Omron Sysmac Studio project SPA_P8_3 (Sysmac Studio 1.23.0.14, StandardProject)

# Controller new_Controller_0: NX1P2-1040DT1 version 1.18
Axis eje_real, settings changed from default: AxisType=ServoType, UnitsConversion=EnumElement2, UnitsNumerator=8380608, UnitsDenominator=143, MaxVelocity=200, MaxJogVelocity=20, HomingMode=BackupAndPressingTime, StartDirection=NegativeDirection, OriginInputDetectionDirection=NegativeDirection, HomingVelocity=200, HomingApproachVelocity=10, OriginCompensationValue=10, CompensationVelocity=10, ModuloMAXPosition=360, ModuloMINPosition=0, EncoderTypes=Abs
Axis eje_virtual, settings changed from default: AxisNumber=1, UnitsConversion=EnumElement2, UnitsNumerator=8380608, UnitsDenominator=143, MaxVelocity=200, MaxJogVelocity=20
Task PrimaryTask (priority 4, period or condition 2000): Programa0

VAR_GLOBAL CONSTANT
    eje_real : _sAXIS_REF;  (* at MC://_MC_AX[0] *)
END_VAR
VAR_GLOBAL
    PM : BOOL;  (* Pulsador Marcha; at BuiltInIO://cpu/#0/Input_Bit_00 *)
    PP : BOOL;  (* Pulsador Paro; at BuiltInIO://cpu/#0/Input_Bit_01 *)
    PR : BOOL;  (* Pulsador Rearme; at BuiltInIO://cpu/#0/Input_Bit_02 *)
    detector_pieza AT %W0.00 : BOOL;  (* Detector simulado de pieza; published *)
    servo_on AT %W0.01 : BOOL;  (* Interruptor de activación de ejes; published *)
END_VAR
VAR_GLOBAL CONSTANT
    eje_virtual : _sAXIS_REF;  (* at MC://_MC_AX[1] *)
END_VAR
VAR_GLOBAL
    pm_hmi AT %W0.02 : BOOL;  (* Marcha HMI; published *)
    pr_hmi AT %W0.03 : BOOL;  (* Rearme HMI; published *)
    pp_hmi AT %W0.04 : BOOL;  (* Paro HMI; published *)
    pm_var : BOOL;  (* Variable Marcha *)
    pr_var : BOOL;  (* Variable Rearme *)
    pp_var : BOOL;  (* Variable Paro *)
END_VAR
VAR_GLOBAL RETAIN
    piezas_cortadas AT %D0 : INT;  (* Número de piezas cortadas; published *)
END_VAR
VAR_GLOBAL
    detector_negativo : BOOL;  (* Detector de límite negativo; at ECAT://node#2/Digital inputs/NOT *)
    detector_positivo : BOOL;  (* Detector de límite positivo; at ECAT://node#2/Digital inputs/POT *)
    selector_pieza AT %W0.05 : BOOL;  (* ON: 20cm / OFF: 10cm; published *)
END_VAR

PROGRAM Programa0
VAR
    reset_eje_real : MC_Reset;
    power_eje_real : MC_Power;
    home_eje_real : MC_Home;
    etapa_produccion : SINT := 0;  (* Etapa actual grafcet principal *)
    etapa_activar : SINT := 0;  (* Etapa actual grafcet activación *)
    reset_eje_virtual : MC_Reset;
    power_eje_virtual : MC_Power;
    home_eje_virtual : MC_Home;
    inicio_corte : MC_MoveAbsolute;
    grosor_corte : LREAL;  (* Grosor del corte en mm *)
    avance_pieza : MC_MoveRelative;
    retroceso_cinta : MC_MoveZeroPosition;
    corte : MC_MoveRelative;
    MC_inicio_corte : MC_MoveAbsolute;
    MC_corte : MC_MoveRelative;
    cortes_realizados : CTU;
    etapa_paro : SINT;  (* Etapa actual grafcet paro *)
    rearme_cinta : MC_MoveZeroPosition;
    rearme_cortadora : MC_MoveZeroPosition;
    retroceso_cortadora : MC_MoveZeroPosition;
    avance_corte : MC_MoveRelative;
    retroceso_corte : MC_MoveRelative;
    paro_eje_real : MC_Stop;
    paro_eje_virtual : MC_Stop;
    reset_eje_real_paro : MC_Reset;
    reset_eje_virtual_paro : MC_Reset;
    tiempo : BOOL;
    status : _sTimer;
END_VAR
VAR RETAIN
    n_cortes : INT;  (* Número de cortes realizados *)
END_VAR
VAR
    avance_pieza_final : MC_MoveRelative;
    grosor_pieza : LREAL;  (* Grosor de la pieza en mm *)
    grosor_corte_negativo : LREAL;  (* Grosor del corte invertido *)
END_VAR
VAR_EXTERNAL CONSTANT
    eje_real : _sAXIS_REF;
END_VAR
VAR_EXTERNAL
    PM : BOOL;
    servo_on : BOOL;
END_VAR
VAR_EXTERNAL CONSTANT
    eje_virtual : _sAXIS_REF;
END_VAR
VAR_EXTERNAL
    detector_pieza : BOOL;
    PP : BOOL;
    PR : BOOL;
    pm_var : BOOL;
    pm_hmi : BOOL;
    pp_var : BOOL;
    pp_hmi : BOOL;
    pr_var : BOOL;
    pr_hmi : BOOL;
    detector_negativo : BOOL;
    detector_positivo : BOOL;
    selector_pieza : BOOL;
    piezas_cortadas : INT;
END_VAR
VAR
    _p1 : BOOL;
    _e2 : R_TRIG;
    _t3 : BOOL;
END_VAR

(* Section activar: ladder, written here as Structured Text *)

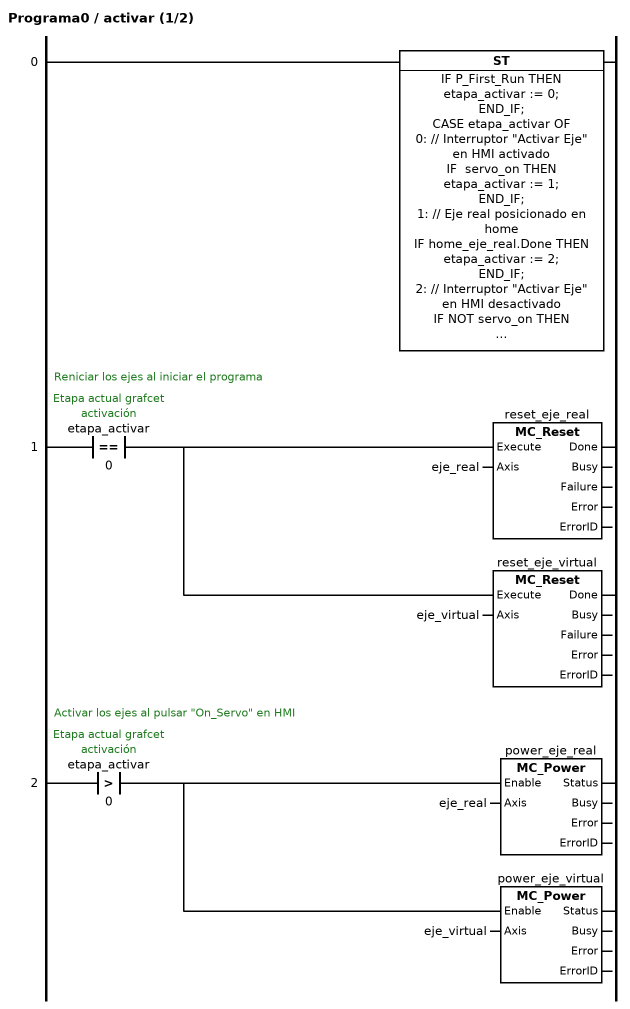
(* Rung 0 *)
IF P_First_Run THEN
	etapa_activar := 0;
END_IF;

CASE etapa_activar OF
	0: // Interruptor "Activar Eje" en HMI activado
		IF  servo_on THEN
			etapa_activar := 1;
		END_IF;
	1: // Eje real posicionado en home
		IF home_eje_real.Done THEN
			etapa_activar := 2;
		END_IF;
	2: // Interruptor "Activar Eje" en HMI desactivado
		IF NOT servo_on THEN
			etapa_activar := 0;
		END_IF;
END_CASE;
(* Rung 1: Reniciar los ejes al iniciar el programa *)
reset_eje_real(Execute := etapa_activar = 0, Axis := eje_real);
reset_eje_virtual(Execute := etapa_activar = 0, Axis := eje_virtual);
(* Rung 2: Activar los ejes al pulsar "On_Servo" en HMI *)
power_eje_real(Enable := etapa_activar > 0, Axis := eje_real);
power_eje_virtual(Enable := etapa_activar > 0, Axis := eje_virtual);

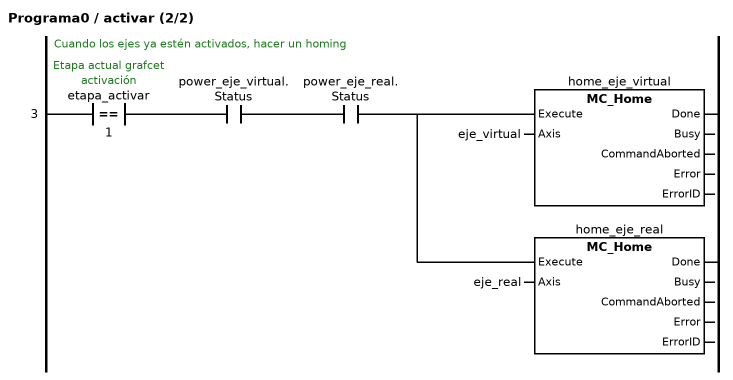
(* Rung 3: Cuando los ejes ya estén activados, hacer un homing *)
_p1 := (etapa_activar = 1) AND power_eje_virtual.Status AND power_eje_real.Status;
home_eje_virtual(Execute := _p1, Axis := eje_virtual);
home_eje_real(Execute := _p1, Axis := eje_real);

(* Section produccion: ladder, written here as Structured Text *)

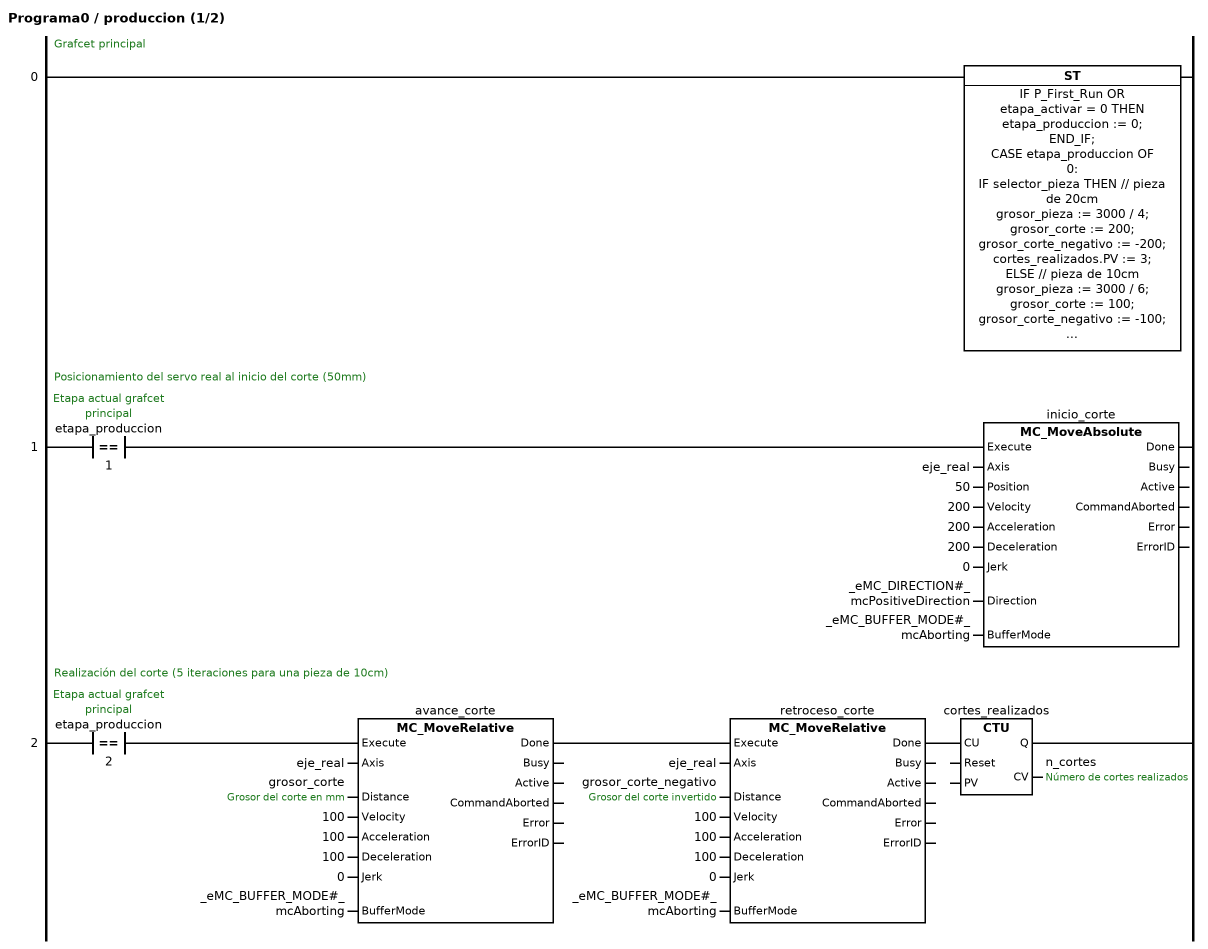
(* Rung 0: Grafcet principal *)
IF P_First_Run OR etapa_activar = 0 THEN
	etapa_produccion := 0;
END_IF;

CASE etapa_produccion OF
    0:
		IF selector_pieza THEN // pieza de 20cm
			grosor_pieza := 3000 / 4;
			grosor_corte := 200;
			grosor_corte_negativo := -200;
			cortes_realizados.PV := 3;
		ELSE // pieza de 10cm
			grosor_pieza := 3000 / 6;
			grosor_corte := 100;
			grosor_corte_negativo := -100;
			cortes_realizados.PV := 5;
		END_IF;
		cortes_realizados.Reset := TRUE;
		// los servos están iniciados y se pulsa marcha
		IF pm_var AND etapa_activar = 2 AND etapa_paro = 0 THEN
			piezas_cortadas := 0;
			cortes_realizados.Reset := FALSE;
			etapa_produccion := 1;
		END_IF;
	1: // el servo real está en posición de inicio de corte (50mm)
		// y se hay pieza en posición de corte
		IF inicio_corte.Done AND detector_pieza THEN
			etapa_produccion := 2;
		END_IF;
	2: // ya se ha realizado el corte de la pieza
		IF retroceso_corte.Done THEN
			piezas_cortadas := piezas_cortadas + 1;
			etapa_produccion := 3;
		END_IF;
	3: // la pieza ya ha avanzado a la posición de corte
		IF cortes_realizados.Q THEN // ya se han realizado todos los cortes
			piezas_cortadas := piezas_cortadas + 1;
			etapa_produccion := 4;
		ELSIF avance_pieza.Done THEN // no se han realizado todos los cortes
			etapa_produccion := 1;
		END_IF;
	4: // la cinta ya ha vuelto al inicio
		IF retroceso_cinta.Done THEN
			etapa_produccion := 0;
		END_IF;
END_CASE;
(* Rung 1: Posicionamiento del servo real al inicio del corte (50mm) *)
inicio_corte(Execute := etapa_produccion = 1, Axis := eje_real, Position := 50, Velocity := 200, Acceleration := 200, Deceleration := 200, Jerk := 0, Direction := _eMC_DIRECTION#_mcPositiveDirection, BufferMode := _eMC_BUFFER_MODE#_mcAborting);
(* Rung 2: Realización del corte (5 iteraciones para una pieza de 10cm) *)
avance_corte(Execute := etapa_produccion = 2, Axis := eje_real, Distance := grosor_corte, Velocity := 100, Acceleration := 100, Deceleration := 100, Jerk := 0, BufferMode := _eMC_BUFFER_MODE#_mcAborting);
retroceso_corte(Execute := avance_corte.Done, Axis := eje_real, Distance := grosor_corte_negativo, Velocity := 100, Acceleration := 100, Deceleration := 100, Jerk := 0, BufferMode := _eMC_BUFFER_MODE#_mcAborting);
_e2(CLK := retroceso_corte.Done);
cortes_realizados(CU := _e2.Q, CV => n_cortes);

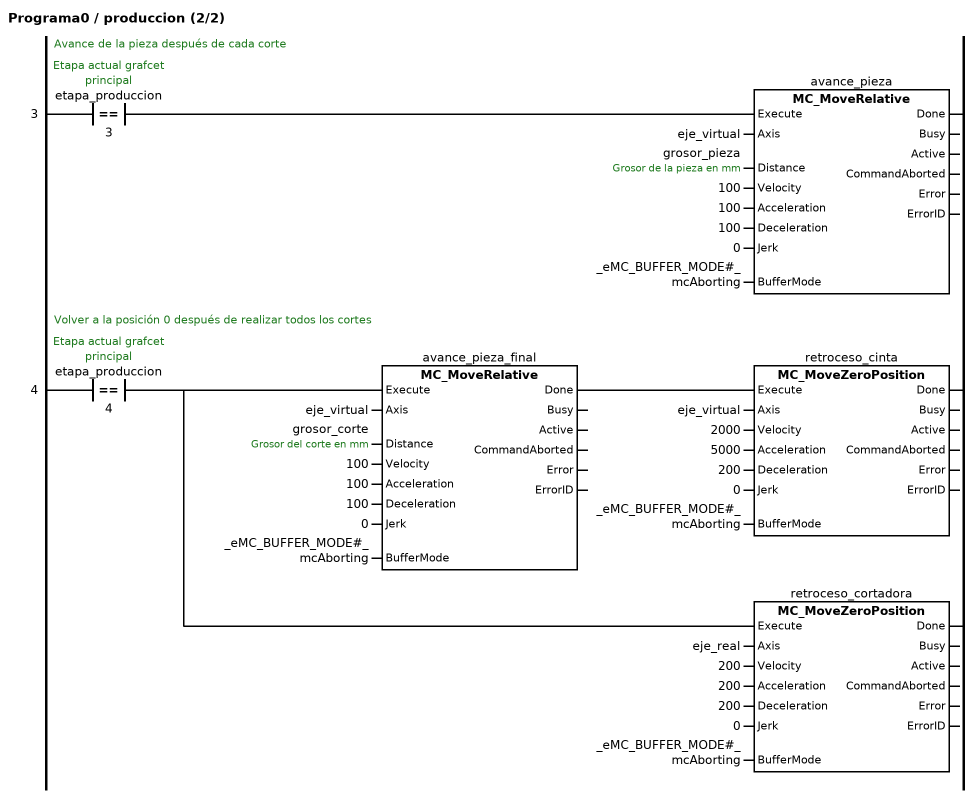
(* Rung 3: Avance de la pieza después de cada corte *)
avance_pieza(Execute := etapa_produccion = 3, Axis := eje_virtual, Distance := grosor_pieza, Velocity := 100, Acceleration := 100, Deceleration := 100, Jerk := 0, BufferMode := _eMC_BUFFER_MODE#_mcAborting);
(* Rung 4: Volver a la posición 0 después de realizar todos los cortes *)
avance_pieza_final(Execute := etapa_produccion = 4, Axis := eje_virtual, Distance := grosor_corte, Velocity := 100, Acceleration := 100, Deceleration := 100, Jerk := 0, BufferMode := _eMC_BUFFER_MODE#_mcAborting);
retroceso_cinta(Execute := avance_pieza_final.Done, Axis := eje_virtual, Velocity := 2000, Acceleration := 5000, Deceleration := 200, Jerk := 0, BufferMode := _eMC_BUFFER_MODE#_mcAborting);
retroceso_cortadora(Execute := etapa_produccion = 4, Axis := eje_real, Velocity := 200, Acceleration := 200, Deceleration := 200, Jerk := 0, BufferMode := _eMC_BUFFER_MODE#_mcAborting);

(* Section paro: ladder, written here as Structured Text *)

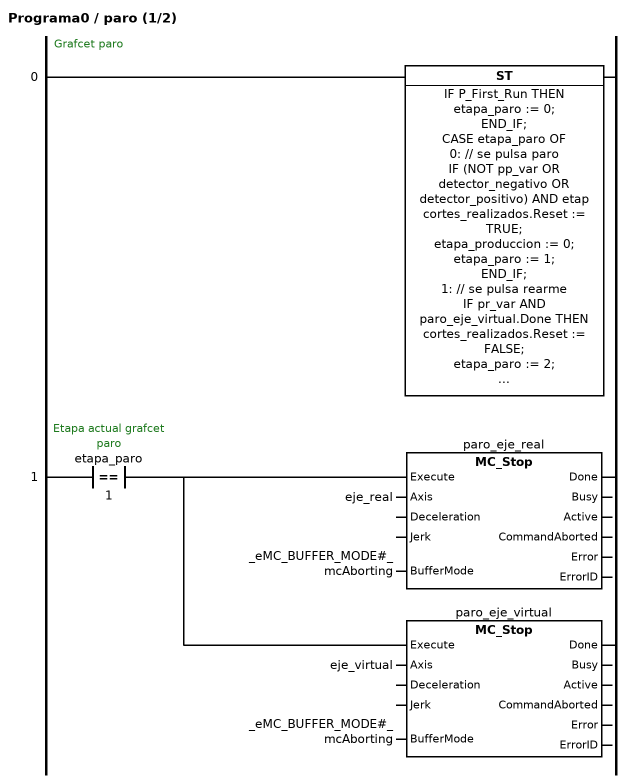
(* Rung 0: Grafcet paro *)
IF P_First_Run THEN
	etapa_paro := 0;
END_IF;

CASE etapa_paro OF
	0: // se pulsa paro
		IF (NOT pp_var OR detector_negativo OR detector_positivo) AND etapa_activar = 2 THEN
			cortes_realizados.Reset := TRUE;
			etapa_produccion := 0;
			etapa_paro := 1;
		END_IF;
	1: // se pulsa rearme
		IF pr_var AND paro_eje_virtual.Done THEN
			cortes_realizados.Reset := FALSE;
			etapa_paro := 2;
		END_IF;
	2: // los dos ejes ya están en posición 0
		IF rearme_cinta.Done AND rearme_cortadora.Done THEN
			etapa_paro := 0;
		END_IF;
END_CASE;
(* Rung 1 *)
paro_eje_real(Execute := etapa_paro = 1, Axis := eje_real, BufferMode := _eMC_BUFFER_MODE#_mcAborting);
paro_eje_virtual(Execute := etapa_paro = 1, Axis := eje_virtual, BufferMode := _eMC_BUFFER_MODE#_mcAborting);

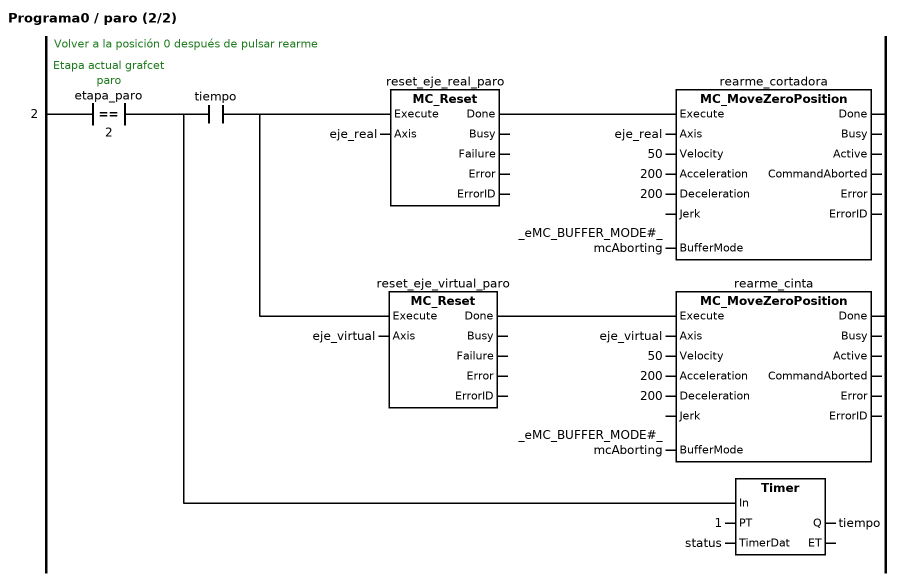
(* Rung 2: Volver a la posición 0 después de pulsar rearme *)
reset_eje_real_paro(Execute := (etapa_paro = 2) AND tiempo, Axis := eje_real);
rearme_cortadora(Execute := reset_eje_real_paro.Done, Axis := eje_real, Velocity := 50, Acceleration := 200, Deceleration := 200, BufferMode := _eMC_BUFFER_MODE#_mcAborting);
reset_eje_virtual_paro(Execute := (etapa_paro = 2) AND tiempo, Axis := eje_virtual);
rearme_cinta(Execute := reset_eje_virtual_paro.Done, Axis := eje_virtual, Velocity := 50, Acceleration := 200, Deceleration := 200, BufferMode := _eMC_BUFFER_MODE#_mcAborting);
_t3 := Timer(In := etapa_paro = 2, PT := 1, TimerDat := status, Q => tiempo);

(* Section hmi_plc: ladder, written here as Structured Text *)

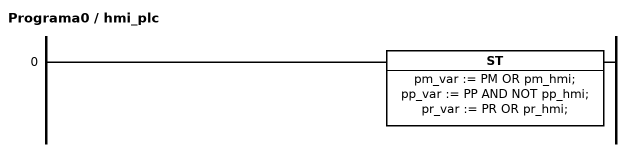
(* Rung 0 *)
pm_var := PM OR pm_hmi;
pp_var := PP AND NOT pp_hmi;
pr_var := PR OR pr_hmi;
END_PROGRAM